// TIA Portal V19 export
DATA_BLOCK "Config"   // DB61
// stored: Access Published, MemoryReserve 100, Namespace Unit3.EM1
   VAR
      em { ExternalWritable := 'False'} : "LAF_typeEmConfiguration";   // Configuration of EM Parameters
      axis { ExternalWritable := 'False'} : Array[1.._.U3EM1_NO_OF_AXES] of DB_ANY;   // Assign the axis of the EM
      em1Parameters : "LAF_typeNgConveyorEm1Parameters";
   END_VAR
BEGIN
   em.referenceDesignator.parent := WSTRING#'U1';
   em.referenceDesignator.relative := WSTRING#'EM1';
   em1Parameters.cm2Axis111.production.distanceList[0].position := 300.0;
END_DATA_BLOCK
